// TwinCAT 3 PLC project TcoAimTtiPowerSupply
// Title: TcoAimTtiPowerSupply
// Company: Vortex.Library
// Author: TcOpenGroup
// ProjectVersion: 0.6.0.913
// ProgramVersion: 3.1.4024.12
// libraries:
//   Tc2_MC2, * (Beckhoff Automation GmbH)
//   Tc2_MC2_Drive, * (Beckhoff Automation GmbH)
//   Tc2_Standard, * (Beckhoff Automation GmbH)
//   Tc2_System, * (Beckhoff Automation GmbH)
//   Tc3_Module, * (Beckhoff Automation GmbH)
//   TcoAbstractions, 0.6.0.913 (Vortex.Library)
//   TcoCore, 0.6.0.913 (Vortex.Library)
//   TcoIo, 0.6.0.913 (Vortex.Library)
//   TcoUtilities, 0.6.0.913 (Vortex.Library)
// project tree:
//   DUTs/ TcoQlSeriesSupply_Config_v_1_x_x.TcDUT, TcoQlSeriesSupply_GetControl_v_1_x_x.TcDUT, TcoQlSeriesSupply_SetControl_v_1_x_x.TcDUT, TcoQlSeriesSupply_State_v_1_x_x.TcDUT, TcoQlSeriesSupply_Status_v_1_x_x.TcDUT
//   / PlcTask.TcTTO
//   POUs/ MAIN.TcPOU
//   POUs/Prototypes/Command/ TcoQlGetCommandTask.TcPOU, TcoQlSetCommandTask.TcPOU, TcoQlSeriesSupplyTask.TcPOU
//   POUs/Prototypes/QLSeries/ TcoQl355P_v_1_x_x.TcPOU
//   POUs/Prototypes/Structs/ eTcoQWlSeriesSupplyGetCommands_v_1_x_x.TcDUT, eTcoQWlSeriesSupplySetCommands_v_1_x_x.TcDUT
// real-time tasks:
//   TASK PlcTask: cycle T#10ms, priority 20, ADS port 350
//   TASK PlcTask1: cycle T#10ms, priority 1, ADS port 351
//   TASK PN: cycle T#8ms, priority 2, ADS port 301
// motion (NC):
//   TASK NC-Task 1 SAF: cycle T#2ms, priority 4, ADS port 501
//   TASK NC-Task 1 SVB: cycle T#10ms, priority 8, ADS port 511
//   AXIS Axis 1 (id 1)
//     Dynamic: Acceleration=5979.5, Deceleration=5979.5, Jerk=17938.5
//     Velo: RefSearch=39.8633642666667, RefSync=39.8633642666667, SlowManual=199.316821333333, FastManual=1195.900928, Fast=3986.33642666667, Maximum=3986.34
//     OtherSettings: AllowMotionCmdToSlave=true
//     encoder EncType=1
//       EncPara: ScaleFactorNumerator=104.8576, ScaleFactorDenominator=1048576, Offset=-0.001200000000608
//     drive DrvType=5
//       Analog: VeloReferenz=4384.97006933333, TorqueSetpointScale=10, ScaleFactorActTorque=0.1
//       TimeComp: TaskDelayCycles=1
//     controller CtrType=1
//       CtrPara: PriorControlFactor=1
//         Observer: BandWidth=20
//   AXIS Axis 2 (id 2)
//     Dynamic: Acceleration=500, Deceleration=500, Jerk=1000
//     Velo: SlowManual=10, FastManual=50, Maximum=3986.34
//     OtherSettings: AllowMotionCmdToSlave=true
//     encoder EncType=1
//       EncPara: ScaleFactorNumerator=1, ScaleFactorDenominator=1024
//     drive DrvType=5
//       Analog: VeloReferenz=4384.97006933333, TorqueSetpointScale=10, ScaleFactorActTorque=0.1
//       TimeComp: TaskDelayCycles=1
//     controller CtrType=1
//       CtrPara: PriorControlFactor=1
//         PosDiffControl: Enable=false
//         PID: PosKp=0.1
//         Observer: BandWidth=20
//   AXIS Axis 3 (id 3)
//     Dynamic: Acceleration=500, Deceleration=500, Jerk=1000
//     Velo: SlowManual=10, FastManual=50, Maximum=3986.34
//     OtherSettings: AllowMotionCmdToSlave=true
//     encoder EncType=1
//       EncPara: ScaleFactorNumerator=1, ScaleFactorDenominator=1024
//     drive DrvType=5
//       Analog: VeloReferenz=4384.97006933333, TorqueSetpointScale=10, ScaleFactorActTorque=0.1
//       TimeComp: TaskDelayCycles=1
//     controller CtrType=1
//       CtrPara: PriorControlFactor=1
//         PosDiffControl: Enable=false
//         PID: PosKp=0.1
//         Observer: BandWidth=20
//   AXIS Axis 4 (id 4)
//     Dynamic: Acceleration=500, Deceleration=500, Jerk=1000
//     Velo: SlowManual=10, FastManual=50, Maximum=3986.34
//     OtherSettings: AllowMotionCmdToSlave=true
//     encoder EncType=1
//       EncPara: ScaleFactorNumerator=1, ScaleFactorDenominator=1024
//     drive DrvType=5
//       Analog: VeloReferenz=4384.97006933333, TorqueSetpointScale=10, ScaleFactorActTorque=0.1
//       TimeComp: TaskDelayCycles=1
//     controller CtrType=1
//       CtrPara: PriorControlFactor=1
//         PosDiffControl: Enable=false
//         PID: PosKp=0.1
//         Observer: BandWidth=20
// I/O:
//   DEVICE Device 4 (EtherCAT) (disabled), AmsNetId 172.20.10.104.5.1
//     Term 1 (EK1100) [EK1100 EtherCAT Coupler (2A E-Bus)]
//       Term 2 (EL1008) [EL1008 8Ch. Dig. Input 24V, 3ms]
//       Term 3 (EL2008) [EL2008 8Ch. Dig. Output 24V, 0.5A]
//       Term 4 (EL3052) [EL3052 2Ch. Ana. Input 4-20mA]
//       Term 5 (EL9576) [EL9576 Brake chopper terminal]
//       Term 6 (EL7211-0010) [EL7211-0010 1Ch. MDP742 Servo motor output stage with OCT (50V, 4.5A RMS)]
//       Term 14 (EL7047) [EL7047 1Ch. Stepper motor output stage (50V, 5A)]
//       Term 8 (EL9011) [EL9011 End Terminal]
//   DEVICE Device 1 (EtherCAT) (disabled), AmsNetId 192.168.4.1.2.1
//     Drive 7 (IndraDrive MPB20) [IndraDrive MPB20]
//   DEVICE Device 2 (EtherCAT) (disabled), AmsNetId 192.168.4.1.3.1
//     Term 1 (EK1200) [EK1200-5000 EtherCAT Power supply (2A E-Bus)]
//       Term 10 (EK1122) [EK1122 2 port EtherCAT junction]
//       Term 13 (EL6631) [EL6631 PROFINET IO Controller]
//       Term 12 (EL1809) [EL1809 16Ch. Dig. Input 24V, 3ms]
//       Term 13 (EL2809) [EL2809 16Ch. Dig. Output 24V, 0.5A]
//       Term 15 (EL4004) [EL4004 4Ch. Ana. Output 0-10V, 12bit]
//       Term 16 (EL7342) [EL7342 2Ch. DC motor output stage (50V, 3.5A)]
//       Term 17 (EL4004) [EL4004 4Ch. Ana. Output 0-10V, 12bit]
//       Term 18 (EL6001) [EL6001 Interface (RS232)]
//       Term 10 (EL9011) [EL9011 End Terminal]
//   DEVICE Device 3 (EL6631) (disabled), AmsNetId 192.168.4.1.4.1
//     robot1 [ABB Robotics The robot controller's internal PROFINET IO device. 888-3] (disabled)
//       modules: Term 1 (DAP Module), Term 2 (DI 64 bytes), Term 3 (DO 64 bytes)
//     robot2 [ABB Robotics The OmniCore controller's internal PROFINET IO device. 3020-x]
//       modules: Term 7 (DAP Module), Term 8 (DI 64 bytes), Term 9 (DO 64 bytes)

CONFIGURATION TcoAimTtiPowerSupply
    RESOURCE PLC ON TwinCAT3
        TASK PlcTask(INTERVAL := T#10ms, PRIORITY := 20);
        PROGRAM MAIN WITH PlcTask : MAIN;
    END_RESOURCE
END_CONFIGURATION

// ---- DUTs/TcoQlSeriesSupply_Config_v_1_x_x.TcDUT
TYPE TcoQlSeriesSupply_Config_v_1_x_x :
STRUCT
    InfoTime : TIME := T#2S;
    ErrorTime : TIME := T#0S;
    IpAddress : STRING;
    Port : UINT := 9221;
    Timeout : UINT := 1000;
END_STRUCT
END_TYPE

// ---- DUTs/TcoQlSeriesSupply_GetControl_v_1_x_x.TcDUT
TYPE TcoQlSeriesSupply_GetControl_v_1_x_x :
STRUCT
    Command : eTcoQWlSeriesSupplyGetCommands_v_1_x_x;
    {attribute addProperty Name "<#Nvalue#>"}
    NValue : USINT; //The number of the output or status register to which the command relates.
//Note that on single output supplies <N>=1 always.
//Note also that <N>= 3 refers to the AUX output. The AUX output has limited remote
//control functionality. For clarity, the commands where <N>= 3 can be used are
//explicitly commented; elsewhere only <N>= 1 or <N>= 2 can be used.
END_STRUCT
END_TYPE

// ---- DUTs/TcoQlSeriesSupply_SetControl_v_1_x_x.TcDUT
TYPE TcoQlSeriesSupply_SetControl_v_1_x_x :
STRUCT
    Command : eTcoQWlSeriesSupplySetCommands_v_1_x_x;
    {attribute addProperty Name "<#NRF#>"}
    NrfValue : REAL; //A number in any format. e.g. 12, 12·00, 1·2 e1 and 120 e-1 are all accepted as the
    //number 12. Any number, when received, is converted to the required precision
    //consistent with the use then rounded up to obtain the value of the command.
    {attribute addProperty Name "<#Nvalue#>"}
    NValue : USINT := 1; //The number of the output or status register to which the command relates.
//Note that on single output supplies <N>=1 always.
//Note also that <N>= 3 refers to the AUX output. The AUX output has limited remote
//control functionality. For clarity, the commands where <N>= 3 can be used are
//explicitly commented; elsewhere only <N>= 1 or <N>= 2 can be used.
END_STRUCT
END_TYPE

// ---- DUTs/TcoQlSeriesSupply_State_v_1_x_x.TcDUT
TYPE TcoQlSeriesSupply_State_v_1_x_x :
STRUCT
    {attribute addProperty Name "<#Raw Response#>"}
    Resposne : STRING(255);
    {attribute addProperty Name "<#NR1#>"}
    Nr1Value : INT; //<NR1> A number with no fractional part, i.e. an integer.
    {attribute addProperty Name "<#NR2#>"}
    Nr2Value : REAL; //<NR2> A number in fixed point format e.g. 11·52, 0·78 etc.
    {attribute addProperty Name "<#N #>"}
    NValue : USINT; //The number of the output or status register to which the command relates.
    //Note that on single output supplies <N>=1 always.
    //Note also that <N>= 3 refers to the AUX output. The AUX output has limited remote
    //control functionality. For clarity, the commands where <N>= 3 can be used are
    //explicitly commented; elsewhere only <N>= 1 or <N>= 2 can be used.
    {attribute addProperty Name "<#Convert Message#>"}
    ConvertMessage : STRING;
END_STRUCT
END_TYPE

// ---- DUTs/TcoQlSeriesSupply_Status_v_1_x_x.TcDUT
TYPE TcoQlSeriesSupply_Status_v_1_x_x :
STRUCT
    ActionDescription : STRING(100);
    State : TcoQlSeriesSupply_State_v_1_x_x;
END_STRUCT
END_TYPE

// ---- POUs/Prototypes/Structs/eTcoQWlSeriesSupplyGetCommands_v_1_x_x.TcDUT
{attribute 'qualified_only'}
{attribute 'strict'}
TYPE eTcoQWlSeriesSupplyGetCommands_v_1_x_x :
(
    //Instrument Specific Commands
    V := 1,
    I := 2,
    OVP := 3,
    OCP := 4,
    VO := 5,
    IO := 6,
    RANGE := 7,
    DELTAV := 8,
    DELTAI := 9,
    OP := 10,
    LSR := 11,
    LSE := 12,
    //System and Status Commands
    EER := 22,
    QER := 23,
    ESE := 24,
    ESR := 25,
    IST := 26,
    OPC := 27,
    PRE := 28,
    SRE := 29,
    STB := 30,
    //Interface Management Commands
    IFLOCK := 41,
    ADDRESS := 42,
    IPADDR := 43,
    NETMASK := 44,
    NETCONFIG := 45,
    //Miscellaneous Commands
    IDN := 70,
    TST := 71
);
END_TYPE

// ---- POUs/Prototypes/Structs/eTcoQWlSeriesSupplySetCommands_v_1_x_x.TcDUT
{attribute 'qualified_only'}
{attribute 'strict'}
TYPE eTcoQWlSeriesSupplySetCommands_v_1_x_x :
(
    //Instrument Specific Commands
    V := 1,
    V_Verif := 2,
    OVP := 3,
    I := 4,
    OCP := 5,
    RANGE := 6,
    DELTAV := 7,
    DELTAI := 8,
    INCV := 9,
    INCV_Verif := 10,
    DECV := 11,
    DECV_Verif := 12,
    INCI := 13,
    DECI := 14,
    OP := 15,
    OPALL := 16,
    SENSE := 17,
    MODE := 18,
    TRIPRST := 19,
    LSE := 21,
    SAV := 22,
    RCL := 23,
    //System and Status Commands
    RST := 24,
    CLS := 25,
    ESE := 26,
    OPC := 27,
    PRE := 28,
    SRE := 29,
    WAI := 30,
    //Interface Management Commands
    IFLOCK := 31,
    IFUNLOCK := 32,
    LOCAL := 33,
    NETCONFIG := 34,
    IPADDR := 35,
    NETMASK := 36,
    TRG := 37
);
END_TYPE

// ---- POUs/MAIN.TcPOU
PROGRAM MAIN
VAR
END_VAR

END_PROGRAM

// ---- POUs/Prototypes/Command/TcoQlGetCommandTask.TcPOU
FUNCTION_BLOCK TcoQlGetCommandTask EXTENDS TcoQlSeriesSupplyTask
VAR
    _command : TcoQlSeriesSupply_GetControl_v_1_x_x;
END_VAR

SUPER^(inoConfig := inoConfig, inoStatus := inoStatus);

(*~
    <docu>
        <summary>
            Restores this instance to the Ready state. Can be called explicitly or from within one of the restore mechanisms.
            <para>
                See also <see cref="PlcDocu.TcoCore.TcoTask.AutoRestorable()"/>
            </para>
        </summary>
    </docu>
~*)
METHOD Restore : ITcoRestorable
SUPER^.Restore();
END_METHOD

METHOD WithParams : REFERENCE TO TcoQlGetCommandTask
VAR_INPUT
    inCommand : TcoQlSeriesSupply_GetControl_v_1_x_x;
END_VAR
THIS^._command := inCommand;
WithParams REF= THIS^;
END_METHOD

END_FUNCTION_BLOCK

// ---- POUs/Prototypes/Command/TcoQlSeriesSupplyTask.TcPOU
FUNCTION_BLOCK PUBLIC TcoQlSeriesSupplyTask EXTENDS TcoCore.TcoRemoteTask
VAR_IN_OUT
    inoConfig : TcoQlSeriesSupply_Config_v_1_x_x;
    inoStatus : TcoQlSeriesSupply_Status_v_1_x_x;
END_VAR
VAR
    _errorMessage : TcoCore.TcoMessenger(THIS^);
    {attribute 'hide'}
    _progress : INT := 0;
    {attribute 'hide'}
    _infoTimer : TON;
    {attribute 'hide'}
    _errorTimer : TON;
    {attribute 'hide'}
    _timer : TON;
    {attribute 'hide'}
    _varInfo : __SYSTEM.VAR_INFO;
    {attribute 'hide'}
    _sb : TcoCore.StringBuilder;
END_VAR

SUPER^();

METHOD CallTimers
VAR_INPUT
    inValue : BOOL;
END_VAR
IF __ISVALIDREF(inoConfig) AND THIS^.inoConfig.ErrorTime <> T#0S OR NOT inValue THEN
    _errorTimer(IN := inValue, PT := THIS^.inoConfig.ErrorTime);
END_IF;

IF __ISVALIDREF(inoConfig) AND THIS^.inoConfig.InfoTime <> T#0S OR NOT inValue THEN
    _infoTimer(IN := inValue, PT := THIS^.inoConfig.InfoTime);
END_IF;
END_METHOD

METHOD PROTECTED OnDone
SUPER^.OnDone();

IF __ISVALIDREF(inoStatus) THEN
    THIS^.inoStatus.ActionDescription := '<#Command finished sucessfully.#>';
END_IF;
END_METHOD

(*~
    <docu>
        <summary>
            Executes when task reaches the ```Error``` state.
            <para>
                Do not confuse with <see cref="PlcDocu.TcoCore.TcoTask.WhileError()"/>, that is called cyclically until '''Error''' state is left.
            </para>
        </summary>
    </docu>
~*)
METHOD PROTECTED OnError
VAR
    description : STRING;
END_VAR
SUPER^.OnError();
description := '<#Command finished with error.#>';

IF __ISVALIDREF(inoStatus) THEN
    THIS^.inoStatus.ActionDescription := description;
END_IF;

THIS^._errorMessage.Error(_sb.Clear().Append(description).Append(' To restore acknowledge this alarm.').ToString()).Pin();
END_METHOD

METHOD PROTECTED OnStart
SUPER^.OnStart();

IF __ISVALIDREF(inoStatus) THEN
    THIS^.inoStatus.ActionDescription := '<#Command started.#>';
END_IF;
END_METHOD

(*~
    <docu>
        <summary>
            Restores this instance to the Ready state. Can be called explicitly or from within one of the restore mechanisms.
            <para>
                See also <see cref="PlcDocu.TcoCore.TcoTask.AutoRestorable()"/>
            </para>
        </summary>
    </docu>
~*)
METHOD Restore : ITcoRestorable
SUPER^.Restore();
_progress := 0;
_timer(In := FALSE);
CallTimers(FALSE);
Messenger.UnPin();
_errorMessage.UnPin();
END_METHOD

END_FUNCTION_BLOCK

// ---- POUs/Prototypes/Command/TcoQlSetCommandTask.TcPOU
FUNCTION_BLOCK TcoQlSetCommandTask EXTENDS TcoQlSeriesSupplyTask
VAR
    _command : TcoQlSeriesSupply_SetControl_v_1_x_x;
END_VAR

SUPER^(inoConfig := inoConfig, inoStatus := inoStatus);

(*~
    <docu>
        <summary>
            Restores this instance to the Ready state. Can be called explicitly or from within one of the restore mechanisms.
            <para>
                See also <see cref="PlcDocu.TcoCore.TcoTask.AutoRestorable()"/>
            </para>
        </summary>
    </docu>
~*)
METHOD Restore : ITcoRestorable
SUPER^.Restore();
END_METHOD

METHOD WithParams : REFERENCE TO TcoQlSetCommandTask
VAR_INPUT
    inCommand : TcoQlSeriesSupply_SetControl_v_1_x_x;
END_VAR
THIS^._command := inCommand;
WithParams REF= THIS^;
END_METHOD

END_FUNCTION_BLOCK

// ---- POUs/Prototypes/QLSeries/TcoQl355P_v_1_x_x.TcPOU
FUNCTION_BLOCK TcoQl355P_v_1_x_x EXTENDS TcoCore.TcoComponent
VAR_INPUT
END_VAR
VAR_OUTPUT
END_VAR
VAR
    {attribute addProperty Name "<#Status#>"}
    _status : TcoQlSeriesSupply_Status_v_1_x_x;
    {attribute addProperty Name "<#Config#>"}
    _config : TcoQlSeriesSupply_Config_v_1_x_x;
    _someTaskIsActive : BOOL;
END_VAR
VAR
    {attribute addProperty Name "<#Get Command#>"}
    _getCommandTask : TcoQlGetCommandTask(THIS^);
    {attribute addProperty Name "<#Set Command#>"}
    _setCommandTask : TcoQlSetCommandTask(THIS^);
    {attribute addProperty Name "<#Restore#>"}
    _restoreTask : TcoCore.TcoTask(THIS^);
END_VAR
VAR
    {attribute 'hide'}
    _sb : TcoCore.StringBuilder;
END_VAR

_getCommandTask(inoConfig := _config, inoStatus := _status);
_setCommandTask(inoConfig := _config, inoStatus := _status);
//*************RESTORE********************
_restoreTask.Enabled := TRUE;

IF _restoreTask.Execute() THEN
    Restore();
    _restoreTask.DoneWhen(TRUE);
    _status.ActionDescription := 'Restored';
END_IF
//****************************************

(*~
    <docu>
        <summary>
            Gets the configuration of the IRC 5.
        </summary>
    </docu>
~*)
PROPERTY Config : REFERENCE TO TcoQlSeriesSupply_Config_v_1_x_x
GET
Config REF= _config;
END_GET
END_PROPERTY

METHOD FB_init : BOOL
VAR_INPUT
    bInitRetains : BOOL; // if TRUE, the retain variables are initialized (warm start / cold start)
    bInCopyCode : BOOL; // if TRUE, the instance afterwards gets moved into the copy code (online change)
    ParentObject : ITcoObject;
END_VAR
END_METHOD

METHOD PUBLIC GetCommand : TcoCore.ITcoTaskStatus
VAR_INPUT
    inCommand : TcoQlSeriesSupply_getControl_v_1_x_x;
END_VAR
GetCommand := _getCommandTask.WithParams(inCommand).Invoke();
END_METHOD

PROPERTY GetCommandTask : TcoCore.ITcoTaskStatus
GET
GetCommandTask := _getCommandTask;
END_GET
END_PROPERTY

METHOD PUBLIC GetCurrent : TcoCore.ITcoTaskStatus
VAR_INPUT
    (*~
    <docu>
        <summary>
            The number of the output or status register to which the command relates.
            Note that on single output supplies <N>=1 always.
            Note also that <N>= 3 refers to the AUX output. The AUX output has limited remote control functionality.
            For clarity, the commands where <N>= 3 can be used are explicitly commented; elsewhere only <N>= 1 or <N>= 2 can be used.
        </summary>
    </docu>
    ~*)
    inNValue : USINT;
END_VAR
VAR_OUTPUT
    outCurrent : REAL;
END_VAR
VAR
    command : TcoQlSeriesSupply_GetControl_v_1_x_x;
END_VAR
outCurrent := 0;
command.Command := eTcoQWlSeriesSupplyGetCommands_v_1_x_x.i;
command.NValue := inNValue;
GetCurrent := GetCommand(inCommand := command);

IF GetCurrent.Done THEN
    outCurrent := Status.State.Nr2Value;
END_IF
END_METHOD

METHOD PUBLIC GetOutputIsOff : TcoCore.ITcoTaskStatus
VAR_INPUT
    (*~
    <docu>
        <summary>
            The number of the output or status register to which the command relates.
            Note that on single output supplies <N>=1 always.
            Note also that <N>= 3 refers to the AUX output. The AUX output has limited remote control functionality.
            For clarity, the commands where <N>= 3 can be used are explicitly commented; elsewhere only <N>= 1 or <N>= 2 can be used.
        </summary>
    </docu>
    ~*)
    inNValue : USINT;
END_VAR
VAR_OUTPUT
    outIsOff : BOOL;
END_VAR
VAR
    command : TcoQlSeriesSupply_GetControl_v_1_x_x;
END_VAR
outIsOff := FALSE;
command.Command := eTcoQWlSeriesSupplyGetCommands_v_1_x_x.OP;
command.NValue := inNValue;
GetOutputIsOff := GetCommand(inCommand := command);

IF GetOutputIsOff.Done THEN
    outIsOff := Status.State.Nr2Value = 0;
END_IF
END_METHOD

METHOD PUBLIC GetOutputIsOn : TcoCore.ITcoTaskStatus
VAR_INPUT
    (*~
    <docu>
        <summary>
            The number of the output or status register to which the command relates.
            Note that on single output supplies <N>=1 always.
            Note also that <N>= 3 refers to the AUX output. The AUX output has limited remote control functionality.
            For clarity, the commands where <N>= 3 can be used are explicitly commented; elsewhere only <N>= 1 or <N>= 2 can be used.
        </summary>
    </docu>
    ~*)
    inNValue : USINT;
END_VAR
VAR_OUTPUT
    outIsOn : BOOL;
END_VAR
VAR
    command : TcoQlSeriesSupply_GetControl_v_1_x_x;
END_VAR
outIsOn := FALSE;
command.Command := eTcoQWlSeriesSupplyGetCommands_v_1_x_x.OP;
command.NValue := inNValue;
GetOutputIsOn := GetCommand(inCommand := command);

IF GetOutputIsOn.Done THEN
    outIsOn := Status.State.Nr2Value = 1;
END_IF
END_METHOD

METHOD PUBLIC GetVoltage : TcoCore.ITcoTaskStatus
VAR_INPUT
    (*~
    <docu>
        <summary>
            The number of the output or status register to which the command relates.
            Note that on single output supplies <N>=1 always.
            Note also that <N>= 3 refers to the AUX output. The AUX output has limited remote control functionality.
            For clarity, the commands where <N>= 3 can be used are explicitly commented; elsewhere only <N>= 1 or <N>= 2 can be used.
        </summary>
    </docu>
    ~*)
    inNValue : USINT;
END_VAR
VAR_OUTPUT
    outVoltage : REAL;
END_VAR
VAR
    command : TcoQlSeriesSupply_GetControl_v_1_x_x;
END_VAR
outVoltage := 0;
command.Command := eTcoQWlSeriesSupplyGetCommands_v_1_x_x.V;
command.NValue := inNValue;
GetVoltage := GetCommand(inCommand := command);

IF GetVoltage.Done THEN
    outVoltage := Status.State.Nr2Value;
END_IF
END_METHOD

(*~
    <docu>
        <summary>
            Restores this instance to the Ready state. Can be called explicitly or from within one of the restore mechanisms.
        </summary>
    </docu>
~*)
METHOD Restore : ITcoRestorable
RestoreTasks();
END_METHOD

METHOD INTERNAL RestoreTasks
_getCommandTask.Restore();
_setCommandTask.Restore();
END_METHOD

(*~
    <docu>
        <summary>
            Custom service (manual, maintenance) logic.
            This method must be implemented in derived class.
        </summary>
    </docu>
~*)
METHOD PROTECTED ServiceMode
END_METHOD

METHOD PUBLIC SetCommand : TcoCore.ITcoTaskStatus
VAR_INPUT
    inCommand : TcoQlSeriesSupply_SetControl_v_1_x_x;
END_VAR
SetCommand := _setCommandTask.WithParams(inCommand).Invoke();
END_METHOD

PROPERTY SetCommandTask : TcoCore.ITcoTaskStatus
GET
SetCommandTask := _setCommandTask;
END_GET
END_PROPERTY

METHOD PUBLIC SetCurrent : TcoCore.ITcoTaskStatus
VAR_INPUT
    inCurrent : REAL;
    (*~
    <docu>
        <summary>
            The number of the output or status register to which the command relates.
            Note that on single output supplies <N>=1 always.
            Note also that <N>= 3 refers to the AUX output. The AUX output has limited remote control functionality.
            For clarity, the commands where <N>= 3 can be used are explicitly commented; elsewhere only <N>= 1 or <N>= 2 can be used.
        </summary>
    </docu>
    ~*)
    inNValue : USINT;
END_VAR
VAR
    command : TcoQlSeriesSupply_SetControl_v_1_x_x;
END_VAR
command.Command := eTcoQWlSeriesSupplySetCommands_v_1_x_x.I;
command.NValue := inNValue;
command.NrfValue := inCurrent;
SetCurrent := SetCommand(inCommand := command);
END_METHOD

METHOD PUBLIC SetOutputOff : TcoCore.ITcoTaskStatus
VAR_INPUT
    (*~
    <docu>
        <summary>
            The number of the output or status register to which the command relates.
            Note that on single output supplies <N>=1 always.
            Note also that <N>= 3 refers to the AUX output. The AUX output has limited remote control functionality.
            For clarity, the commands where <N>= 3 can be used are explicitly commented; elsewhere only <N>= 1 or <N>= 2 can be used.
        </summary>
    </docu>
    ~*)
    inNValue : USINT;
END_VAR
VAR
    command : TcoQlSeriesSupply_SetControl_v_1_x_x;
END_VAR
command.Command := eTcoQWlSeriesSupplySetCommands_v_1_x_x.OP;
command.NValue := inNValue;
command.NrfValue := 0;
SetOutputOff := SetCommand(inCommand := command);
END_METHOD

METHOD PUBLIC SetOutputOn : TcoCore.ITcoTaskStatus
VAR_INPUT
    (*~
    <docu>
        <summary>
            The number of the output or status register to which the command relates.
            Note that on single output supplies <N>=1 always.
            Note also that <N>= 3 refers to the AUX output. The AUX output has limited remote control functionality.
            For clarity, the commands where <N>= 3 can be used are explicitly commented; elsewhere only <N>= 1 or <N>= 2 can be used.
        </summary>
    </docu>
    ~*)
    inNValue : USINT;
END_VAR
VAR
    command : TcoQlSeriesSupply_SetControl_v_1_x_x;
END_VAR
command.Command := eTcoQWlSeriesSupplySetCommands_v_1_x_x.OP;
command.NValue := inNValue;
command.NrfValue := 1;
SetOutputOn := SetCommand(inCommand := command);
END_METHOD

METHOD PUBLIC SetVoltage : TcoCore.ITcoTaskStatus
VAR_INPUT
    inVoltage : REAL;
    (*~
    <docu>
        <summary>
            The number of the output or status register to which the command relates.
            Note that on single output supplies <N>=1 always.
            Note also that <N>= 3 refers to the AUX output. The AUX output has limited remote control functionality.
            For clarity, the commands where <N>= 3 can be used are explicitly commented; elsewhere only <N>= 1 or <N>= 2 can be used.
        </summary>
    </docu>
    ~*)
    inNValue : USINT;
END_VAR
VAR
    command : TcoQlSeriesSupply_SetControl_v_1_x_x;
END_VAR
command.Command := eTcoQWlSeriesSupplySetCommands_v_1_x_x.V;
command.NValue := inNValue;
command.NrfValue := inVoltage;
SetVoltage := SetCommand(inCommand := command);
END_METHOD

(*~
    <docu>
        <summary>
            Gets the status of the components.
        </summary>
    </docu>
~*)
PROPERTY Status : REFERENCE TO TcoQlSeriesSupply_Status_v_1_x_x
GET
Status REF= _status;
END_GET
END_PROPERTY

END_FUNCTION_BLOCK
